(* CODESYS project Proj_3Conveyors_-_Codesys_SP19_RECOVERED_2025-03-27T17-36-29.project

Project tree, tasks and I/O mapping:
  Device : CODESYS Control Win V3 x64, 3S - Smart Software Solutions GmbH, version 3.5.19.20
    application Application
      libraries: Standard, 3.5.18.0 (System)
      task MainTask (cyclic, interval t#20ms, priority 1) calls PLC_PRG, SCADA_PRG
      function block Linear_Conveyor [SFC]: passRecipe, copy_recipe
      program PLC_PRG [CFC]
      function block WarehouseInConveyor [SFC]: copy_recipe
      function block Machine [SFC]: IncrementStep, sendTrans, checkOpPossible, copy_recipe, ChangeCurrTool, DefinePassedRecipe
      data type INSTRUCTION
      data type RECIPE_STRUCT
      program SCADA_PRG [ST]
      function block WarehouseOutConveyor [SFC]: copy_recipe
    Ethernet : Ethernet, CODESYS, version 4.2.0.0
      ModbusTCP_Slave_Device : ModbusTCP Slave Device, 3S - Smart Software Solutions GmbH, version 4.3.0.0
          settings: UpdateableHolding = TRUE; DistinctBitAreas = TRUE; Coils Size = 8; Discrete Inputs Size = 8
          output S_sensor1 : BOOL  // Holding Registers.Holding Registers.Bit0
          output S_sensor2 : BOOL  // Holding Registers.Holding Registers.Bit1
          output S_sensor3 : BOOL  // Holding Registers.Holding Registers.Bit2
          output C1_stop : BOOL  // Holding Registers.Holding Registers.Bit0
          output C2_stop : BOOL  // Holding Registers.Holding Registers.Bit1
          output C3_stop : BOOL  // Holding Registers.Holding Registers.Bit2
          output Gate0 : BOOL  // Coils.Coils.Bit0
          output Gate1 : BOOL  // Coils.Coils.Bit1
          output Gate2 : BOOL  // Coils.Coils.Bit2
          unmapped channels: Holding Registers, Input Registers, Coils, Discrete Inputs
      Modbus_TCP_Master : Modbus TCP Master, 3S - Smart Software Solutions GmbH, version 4.3.0.0
          settings: AutoReconnect = TRUE
        Modbus_TCP_Slave : Modbus TCP Slave, 3S - Smart Software Solutions GmbH, version 4.1.0.0
            settings: Unit-ID = 255; IPAddress = [127, 0, 0, 1]; Port = 5502; Channel 0.Function Code = 2; Channel 0.Read Offset = 16#0000; Channel 0.Read Length = 100; Channel 0.Write Offset = 0; Channel 0.Write Length = 0; Channel 0.Cycle Time = 100; Channel 1.Function Code = 15; Channel 1.Read Offset = 0; Channel 1.Read Length = 0; Channel 1.Write Offset = 16#0000; Channel 1.Write Length = 100; Channel 1.Cycle Time = 100
            input  Cin1_Sensor : BOOL  // Channel 0.Channel 0.Bit0
            input  Cin2_Sensor : BOOL  // Channel 0.Channel 0.Bit1
            input  Cin3_Sensor : BOOL  // Channel 0.Channel 0.Bit2
            input  Cin4_Sensor : BOOL  // Channel 0.Channel 0.Bit3
            input  AT1_in0_Sensor : BOOL  // Channel 0.Channel 0.Bit4
            input  AT1_in1_Sensor : BOOL  // Channel 0.Channel 0.Bit5
            input  AT1_in2_Sensor : BOOL  // Channel 0.Channel 0.Bit6
            input  AT1_in3_Sensor : BOOL  // Channel 0.Channel 0.Bit7
            input  AT1_in4_Sensor : BOOL  // Channel 0.Channel 0.Bit0
            input  AT1_out1_Sensor : BOOL  // Channel 0.Channel 0.Bit1
            input  AT1_out2_Sensor : BOOL  // Channel 0.Channel 0.Bit2
            input  AT1_out3_Sensor : BOOL  // Channel 0.Channel 0.Bit3
            input  AT1_out4_Sensor : BOOL  // Channel 0.Channel 0.Bit4
            input  AT1_out5_Sensor : BOOL  // Channel 0.Channel 0.Bit5
            input  AT1_out6_Sensor : BOOL  // Channel 0.Channel 0.Bit6
            input  AT2_out0_Sensor : BOOL  // Channel 0.Channel 0.Bit7
            input  AT2_out1_Sensor : BOOL  // Channel 0.Channel 0.Bit0
            input  AT2_out2_Sensor : BOOL  // Channel 0.Channel 0.Bit1
            input  AT2_out3_Sensor : BOOL  // Channel 0.Channel 0.Bit2
            input  AT2_out4_Sensor : BOOL  // Channel 0.Channel 0.Bit3
            input  AT2_in1_Sensor : BOOL  // Channel 0.Channel 0.Bit4
            input  AT2_in2_Sensor : BOOL  // Channel 0.Channel 0.Bit5
            input  AT2_in3_Sensor : BOOL  // Channel 0.Channel 0.Bit6
            input  AT2_in4_Sensor : BOOL  // Channel 0.Channel 0.Bit7
            input  AT2_in5_Sensor : BOOL  // Channel 0.Channel 0.Bit0
            input  AT2_in6_Sensor : BOOL  // Channel 0.Channel 0.Bit1
            input  Cell0_Ctop_Sensor : BOOL  // Channel 0.Channel 0.Bit2
            input  Cell0_Cmid_Sensor : BOOL  // Channel 0.Channel 0.Bit3
            input  Cell0_Cbot_Sensor : BOOL  // Channel 0.Channel 0.Bit4
            input  Cell1_Mtop_Sensor : BOOL  // Channel 0.Channel 0.Bit5
            input  Cell1_Mtop_Tool_Sensor : BOOL  // Channel 0.Channel 0.Bit6
            input  Cell1_Mtop_Y_minus_Sensor : BOOL  // Channel 0.Channel 0.Bit7
            input  Cell1_Mtop_Y_plus_Sensor : BOOL  // Channel 0.Channel 0.Bit0
            input  Cell1_Mtop_Z_minus_Sensor : BOOL  // Channel 0.Channel 0.Bit1
            input  Cell1_Mtop_Z_plus_Sensor : BOOL  // Channel 0.Channel 0.Bit2
            input  Cell1_Cmid_Sensor : BOOL  // Channel 0.Channel 0.Bit3
            input  Cell1_Mbot_Sensor : BOOL  // Channel 0.Channel 0.Bit4
            input  Cell1_Mbot_Tool_Sensor : BOOL  // Channel 0.Channel 0.Bit5
            input  Cell1_Mbot_Y_minus_Sensor : BOOL  // Channel 0.Channel 0.Bit6
            input  Cell1_Mbot_Y_plus_Sensor : BOOL  // Channel 0.Channel 0.Bit7
            input  Cell1_Mbot_Z_minus_Sensor : BOOL  // Channel 0.Channel 0.Bit0
            input  Cell1_Mbot_Z_plus_Sensor : BOOL  // Channel 0.Channel 0.Bit1
            input  Cell2_Mtop_Sensor : BOOL  // Channel 0.Channel 0.Bit2
            input  Cell2_Mtop_Tool_Sensor : BOOL  // Channel 0.Channel 0.Bit3
            input  Cell2_Mtop_Y_minus_Sensor : BOOL  // Channel 0.Channel 0.Bit4
            input  Cell2_Mtop_Y_plus_Sensor : BOOL  // Channel 0.Channel 0.Bit5
            input  Cell2_Mtop_Z_minus_Sensor : BOOL  // Channel 0.Channel 0.Bit6
            input  Cell2_Mtop_Z_plus_Sensor : BOOL  // Channel 0.Channel 0.Bit7
            input  Cell2_Cmid_Sensor : BOOL  // Channel 0.Channel 0.Bit0
            input  Cell2_Mbot_Sensor : BOOL  // Channel 0.Channel 0.Bit1
            input  Cell2_Mbot_Tool_Sensor : BOOL  // Channel 0.Channel 0.Bit2
            input  Cell2_Mbot_Y_minus_Sensor : BOOL  // Channel 0.Channel 0.Bit3
            input  Cell2_Mbot_Y_plus_Sensor : BOOL  // Channel 0.Channel 0.Bit4
            input  Cell2_Mbot_Z_minus_Sensor : BOOL  // Channel 0.Channel 0.Bit5
            input  Cell2_Mbot_Z_plus_Sensor : BOOL  // Channel 0.Channel 0.Bit6
            input  Cell3_Mtop_Sensor : BOOL  // Channel 0.Channel 0.Bit7
            input  Cell3_Mtop_Tool_Sensor : BOOL  // Channel 0.Channel 0.Bit0
            input  Cell3_Mtop_Y_minus_Sensor : BOOL  // Channel 0.Channel 0.Bit1
            input  Cell3_Mtop_Y_plus_Sensor : BOOL  // Channel 0.Channel 0.Bit2
            input  Cell3_Mtop_Z_minus_Sensor : BOOL  // Channel 0.Channel 0.Bit3
            input  Cell3_Mtop_Z_plus_Sensor : BOOL  // Channel 0.Channel 0.Bit4
            input  Cell3_Cmid_Sensor : BOOL  // Channel 0.Channel 0.Bit5
            input  Cell3_Mbot_Sensor : BOOL  // Channel 0.Channel 0.Bit6
            input  Cell3_Mbot_Tool_Sensor : BOOL  // Channel 0.Channel 0.Bit7
            input  Cell3_Mbot_Y_minus_Sensor : BOOL  // Channel 0.Channel 0.Bit0
            input  Cell3_Mbot_Y_plus_Sensor : BOOL  // Channel 0.Channel 0.Bit1
            input  Cell3_Mbot_Z_minus_Sensor : BOOL  // Channel 0.Channel 0.Bit2
            input  Cell3_Mbot_Z_plus_Sensor : BOOL  // Channel 0.Channel 0.Bit3
            input  Cell4_Mtop_Sensor : BOOL  // Channel 0.Channel 0.Bit4
            input  Cell4_Mtop_Tool_Sensor : BOOL  // Channel 0.Channel 0.Bit5
            input  Cell4_Mtop_Y_minus_Sensor : BOOL  // Channel 0.Channel 0.Bit6
            input  Cell4_Mtop_Y_plus_Sensor : BOOL  // Channel 0.Channel 0.Bit7
            input  Cell4_Mtop_Z_minus_Sensor : BOOL  // Channel 0.Channel 0.Bit0
            input  Cell4_Mtop_Z_plus_Sensor : BOOL  // Channel 0.Channel 0.Bit1
            input  Cell4_Cmid_Sensor : BOOL  // Channel 0.Channel 0.Bit2
            input  Cell4_Mbot_Sensor : BOOL  // Channel 0.Channel 0.Bit3
            input  Cell4_Mbot_Tool_Sensor : BOOL  // Channel 0.Channel 0.Bit4
            input  Cell4_Mbot_Y_minus_Sensor : BOOL  // Channel 0.Channel 0.Bit5
            input  Cell4_Mbot_Y_plus_Sensor : BOOL  // Channel 0.Channel 0.Bit6
            input  Cell4_Mbot_Z_minus_Sensor : BOOL  // Channel 0.Channel 0.Bit7
            input  Cell4_Mbot_Z_plus_Sensor : BOOL  // Channel 0.Channel 0.Bit0
            input  Cell5_Mtop_Sensor : BOOL  // Channel 0.Channel 0.Bit1
            input  Cell5_Mtop_Tool_Sensor : BOOL  // Channel 0.Channel 0.Bit2
            input  Cell5_Mtop_Y_minus_Sensor : BOOL  // Channel 0.Channel 0.Bit3
            input  Cell5_Mtop_Y_plus_Sensor : BOOL  // Channel 0.Channel 0.Bit4
            input  Cell5_Mtop_Z_minus_Sensor : BOOL  // Channel 0.Channel 0.Bit5
            input  Cell5_Mtop_Z_plus_Sensor : BOOL  // Channel 0.Channel 0.Bit6
            input  Cell5_Cmid_Sensor : BOOL  // Channel 0.Channel 0.Bit7
            input  Cell5_Mbot_Sensor : BOOL  // Channel 0.Channel 0.Bit0
            input  Cell5_Mbot_Tool_Sensor : BOOL  // Channel 0.Channel 0.Bit1
            input  Cell5_Mbot_Y_minus_Sensor : BOOL  // Channel 0.Channel 0.Bit2
            input  Cell5_Mbot_Y_plus_Sensor : BOOL  // Channel 0.Channel 0.Bit3
            input  Cell5_Mbot_Z_minus_Sensor : BOOL  // Channel 0.Channel 0.Bit4
            input  Cell5_Mbot_Z_plus_Sensor : BOOL  // Channel 0.Channel 0.Bit5
            input  Cell6_Mtop_Sensor : BOOL  // Channel 0.Channel 0.Bit6
            input  Cell6_Mtop_Tool_Sensor : BOOL  // Channel 0.Channel 0.Bit7
            input  Cell6_Mtop_Y_minus_Sensor : BOOL  // Channel 0.Channel 0.Bit0
            input  Cell6_Mtop_Y_plus_Sensor : BOOL  // Channel 0.Channel 0.Bit1
            input  Cell6_Mtop_Z_minus_Sensor : BOOL  // Channel 0.Channel 0.Bit2
            input  Cell6_Mtop_Z_plus_Sensor : BOOL  // Channel 0.Channel 0.Bit3
            output Cin1_Motor_plus : BOOL  // Channel 1.Channel 1.Bit0
            output Cin1_Motor_minus : BOOL  // Channel 1.Channel 1.Bit1
            output Cin2_Motor_plus : BOOL  // Channel 1.Channel 1.Bit2
            output Cin2_Motor_minus : BOOL  // Channel 1.Channel 1.Bit3
            output Cin3_Motor_plus : BOOL  // Channel 1.Channel 1.Bit4
            output Cin3_Motor_minus : BOOL  // Channel 1.Channel 1.Bit5
            output Cin4_Motor_plus : BOOL  // Channel 1.Channel 1.Bit6
            output Cin4_Motor_minus : BOOL  // Channel 1.Channel 1.Bit7
            output AT1_in0_Motor_plus : BOOL  // Channel 1.Channel 1.Bit0
            output AT1_in0_Motor_minus : BOOL  // Channel 1.Channel 1.Bit1
            output AT1_in0_Warehouse_In : BOOL  // Channel 1.Channel 1.Bit2
            output AT1_in1_Motor_plus : BOOL  // Channel 1.Channel 1.Bit3
            output AT1_in1_Motor_minus : BOOL  // Channel 1.Channel 1.Bit4
            output AT1_in1_Warehouse_In : BOOL  // Channel 1.Channel 1.Bit5
            output AT1_in2_Motor_plus : BOOL  // Channel 1.Channel 1.Bit6
            output AT1_in2_Motor_minus : BOOL  // Channel 1.Channel 1.Bit7
            output AT1_in2_Warehouse_In : BOOL  // Channel 1.Channel 1.Bit0
            output AT1_in3_Motor_plus : BOOL  // Channel 1.Channel 1.Bit1
            output AT1_in3_Motor_minus : BOOL  // Channel 1.Channel 1.Bit2
            output AT1_in3_Warehouse_In : BOOL  // Channel 1.Channel 1.Bit3
            output AT1_in4_Motor_plus : BOOL  // Channel 1.Channel 1.Bit4
            output AT1_in4_Motor_minus : BOOL  // Channel 1.Channel 1.Bit5
            output AT1_in4_Warehouse_In : BOOL  // Channel 1.Channel 1.Bit6
            output AT1_out1_Motor_plus : BOOL  // Channel 1.Channel 1.Bit7
            output AT1_out1_Motor_minus : BOOL  // Channel 1.Channel 1.Bit0
            output AT1_out2_Motor_plus : BOOL  // Channel 1.Channel 1.Bit1
            output AT1_out2_Motor_minus : BOOL  // Channel 1.Channel 1.Bit2
            output AT1_out3_Motor_plus : BOOL  // Channel 1.Channel 1.Bit3
            output AT1_out3_Motor_minus : BOOL  // Channel 1.Channel 1.Bit4
            output AT1_out4_Motor_plus : BOOL  // Channel 1.Channel 1.Bit5
            output AT1_out4_Motor_minus : BOOL  // Channel 1.Channel 1.Bit6
            output AT1_out5_Motor_plus : BOOL  // Channel 1.Channel 1.Bit7
            output AT1_out5_Motor_minus : BOOL  // Channel 1.Channel 1.Bit0
            output AT1_out6_Motor_plus : BOOL  // Channel 1.Channel 1.Bit1
            output AT1_out6_Motor_minus : BOOL  // Channel 1.Channel 1.Bit2
            output AT2_out0_Motor_plus : BOOL  // Channel 1.Channel 1.Bit3
            output AT2_out0_Motor_minus : BOOL  // Channel 1.Channel 1.Bit4
            output AT2_out1_Motor_plus : BOOL  // Channel 1.Channel 1.Bit5
            output AT2_out1_Motor_minus : BOOL  // Channel 1.Channel 1.Bit6
            output AT2_out2_Motor_plus : BOOL  // Channel 1.Channel 1.Bit7
            output AT2_out2_Motor_minus : BOOL  // Channel 1.Channel 1.Bit0
            output AT2_out3_Motor_plus : BOOL  // Channel 1.Channel 1.Bit1
            output AT2_out3_Motor_minus : BOOL  // Channel 1.Channel 1.Bit2
            output AT2_out4_Motor_plus : BOOL  // Channel 1.Channel 1.Bit3
            output AT2_out4_Motor_minus : BOOL  // Channel 1.Channel 1.Bit4
            output AT2_in1_Motor_plus : BOOL  // Channel 1.Channel 1.Bit5
            output AT2_in1_Motor_minus : BOOL  // Channel 1.Channel 1.Bit6
            output AT2_in1_Warehouse_In : BOOL  // Channel 1.Channel 1.Bit7
            output AT2_in2_Motor_plus : BOOL  // Channel 1.Channel 1.Bit0
            output AT2_in2_Motor_minus : BOOL  // Channel 1.Channel 1.Bit1
            output AT2_in2_Warehouse_In : BOOL  // Channel 1.Channel 1.Bit2
            output AT2_in3_Motor_plus : BOOL  // Channel 1.Channel 1.Bit3
            output AT2_in3_Motor_minus : BOOL  // Channel 1.Channel 1.Bit4
            output AT2_in3_Warehouse_In : BOOL  // Channel 1.Channel 1.Bit5
            output AT2_in4_Motor_plus : BOOL  // Channel 1.Channel 1.Bit6
            output AT2_in4_Motor_minus : BOOL  // Channel 1.Channel 1.Bit7
            output AT2_in4_Warehouse_In : BOOL  // Channel 1.Channel 1.Bit0
            output AT2_in5_Motor_plus : BOOL  // Channel 1.Channel 1.Bit1
            output AT2_in5_Motor_minus : BOOL  // Channel 1.Channel 1.Bit2
            output AT2_in5_Warehouse_In : BOOL  // Channel 1.Channel 1.Bit3
            output AT2_in6_Motor_plus : BOOL  // Channel 1.Channel 1.Bit4
            output AT2_in6_Motor_minus : BOOL  // Channel 1.Channel 1.Bit5
            output AT2_in6_Warehouse_In : BOOL  // Channel 1.Channel 1.Bit6
            output Cell0_Ctop_Motor_plus : BOOL  // Channel 1.Channel 1.Bit7
            output Cell0_Ctop_Motor_minus : BOOL  // Channel 1.Channel 1.Bit0
            output Cell0_Cmid_Motor_plus : BOOL  // Channel 1.Channel 1.Bit1
            output Cell0_Cmid_Motor_minus : BOOL  // Channel 1.Channel 1.Bit2
            output Cell0_Cbot_Motor_plus : BOOL  // Channel 1.Channel 1.Bit3
            output Cell0_Cbot_Motor_minus : BOOL  // Channel 1.Channel 1.Bit4
            output Cell1_Mtop_Motor_plus : BOOL  // Channel 1.Channel 1.Bit5
            output Cell1_Mtop_Motor_minus : BOOL  // Channel 1.Channel 1.Bit6
            output Cell1_Mtop_Rotate_minus : BOOL  // Channel 1.Channel 1.Bit7
            output Cell1_Mtop_Rotate_plus : BOOL  // Channel 1.Channel 1.Bit0
            output Cell1_Mtop_Tool : BOOL  // Channel 1.Channel 1.Bit1
            output Cell1_Mtop_Y_minus : BOOL  // Channel 1.Channel 1.Bit2
            output Cell1_Mtop_Y_plus : BOOL  // Channel 1.Channel 1.Bit3
            output Cell1_Mtop_Z_minus : BOOL  // Channel 1.Channel 1.Bit4
            output Cell1_Mtop_Z_plus : BOOL  // Channel 1.Channel 1.Bit5
            output Cell1_Cmid_Motor_plus : BOOL  // Channel 1.Channel 1.Bit6
            output Cell1_Cmid_Motor_minus : BOOL  // Channel 1.Channel 1.Bit7
            output Cell1_Mbot_Motor_plus : BOOL  // Channel 1.Channel 1.Bit0
            output Cell1_Mbot_Motor_minus : BOOL  // Channel 1.Channel 1.Bit1
            output Cell1_Mbot_Rotate_minus : BOOL  // Channel 1.Channel 1.Bit2
            output Cell1_Mbot_Rotate_plus : BOOL  // Channel 1.Channel 1.Bit3
            output Cell1_Mbot_Tool : BOOL  // Channel 1.Channel 1.Bit4
            output Cell1_Mbot_Y_minus : BOOL  // Channel 1.Channel 1.Bit5
            output Cell1_Mbot_Y_plus : BOOL  // Channel 1.Channel 1.Bit6
            output Cell1_Mbot_Z_minus : BOOL  // Channel 1.Channel 1.Bit7
            output Cell1_Mbot_Z_plus : BOOL  // Channel 1.Channel 1.Bit0
            output Cell2_Mtop_Motor_plus : BOOL  // Channel 1.Channel 1.Bit1
            output Cell2_Mtop_Motor_minus : BOOL  // Channel 1.Channel 1.Bit2
            output Cell2_Mtop_Rotate_minus : BOOL  // Channel 1.Channel 1.Bit3
            output Cell2_Mtop_Rotate_plus : BOOL  // Channel 1.Channel 1.Bit4
            output Cell2_Mtop_Tool : BOOL  // Channel 1.Channel 1.Bit5
            output Cell2_Mtop_Y_minus : BOOL  // Channel 1.Channel 1.Bit6
            output Cell2_Mtop_Y_plus : BOOL  // Channel 1.Channel 1.Bit7
            output Cell2_Mtop_Z_minus : BOOL  // Channel 1.Channel 1.Bit0
            output Cell2_Mtop_Z_plus : BOOL  // Channel 1.Channel 1.Bit1
            output Cell2_Cmid_Motor_plus : BOOL  // Channel 1.Channel 1.Bit2
            output Cell2_Cmid_Motor_minus : BOOL  // Channel 1.Channel 1.Bit3
            unmapped channels: Channel 0, Channel 1
*)

// Device/Application/INSTRUCTION
TYPE INSTRUCTION :
STRUCT
	tool: INT;
	process_time: TIME;
END_STRUCT
END_TYPE

// Device/Application/RECIPE_STRUCT
TYPE RECIPE_STRUCT :
STRUCT
	Piece: INT;
	Instruction_list: ARRAY[1..3] OF INSTRUCTION;
	Step: INT;
END_STRUCT
END_TYPE

// Device/Application/PLC_PRG
PROGRAM PLC_PRG
VAR
	C1, C2, C3: Linear_Conveyor;
	M1,M2: Machine;
	WC1: WarehouseInConveyor;
	
	M1_tools : ARRAY[1..3] OF INT := [1,2,3];
	M2_tools : ARRAY[1..3] OF INT := [4,5,6];
	
	test_instruction : INSTRUCTION := (tool := 1, process_time :=T#20S);
	test_instruction2 : INSTRUCTION := (tool := 5, process_time :=T#30S);
	test_array : ARRAY [1..3] OF INSTRUCTION := [test_instruction,test_instruction2,test_instruction];
	
	test_recipe : RECIPE_STRUCT := (Piece:=1, Instruction_list := test_array ,Step:=1);
	
	WCO1: WarehouseOutConveyor;
END_VAR

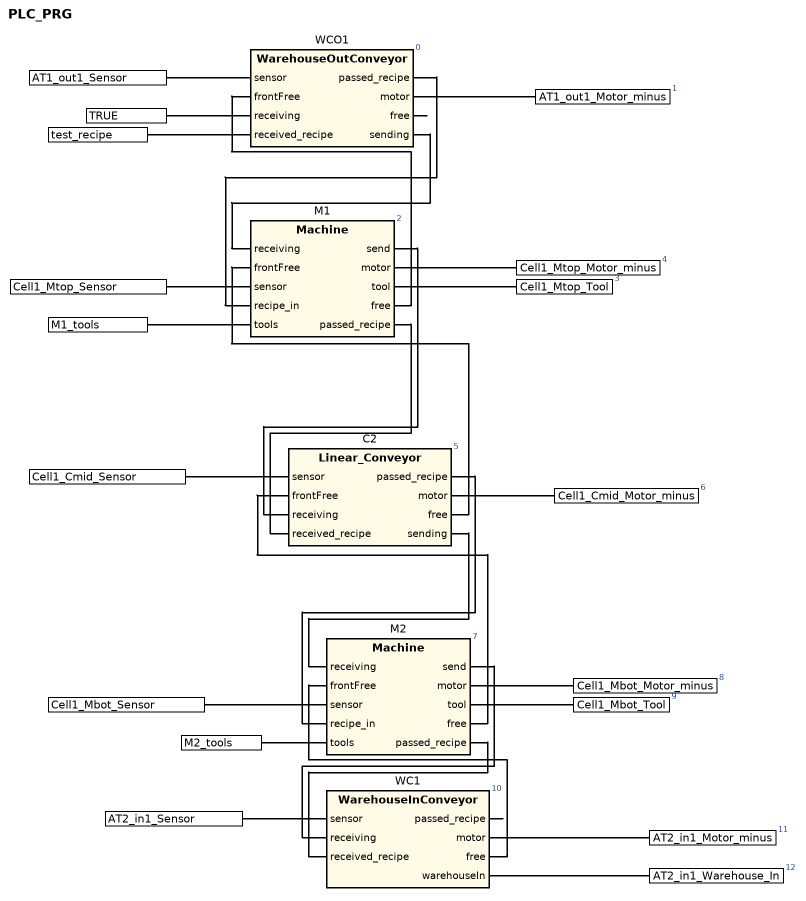
WCO1(sensor := AT1_out1_Sensor, frontFree := M1.free, receiving := TRUE, received_recipe := test_recipe); // WarehouseOutConveyor
AT1_out1_Motor_minus := WCO1.motor;
M1(
    receiving := WCO1.sending,
    frontFree := C2.free,
    sensor := Cell1_Mtop_Sensor,
    recipe_in := WCO1.passed_recipe,
    tools := M1_tools); // Machine
Cell1_Mtop_Tool := M1.tool;
Cell1_Mtop_Motor_minus := M1.motor;
C2(
    sensor := Cell1_Cmid_Sensor,
    frontFree := M2.free,
    receiving := M1.send,
    received_recipe := M1.passed_recipe); // Linear_Conveyor
Cell1_Cmid_Motor_minus := C2.motor;
M2(
    receiving := C2.sending,
    frontFree := WC1.free,
    sensor := Cell1_Mbot_Sensor,
    recipe_in := C2.passed_recipe,
    tools := M2_tools); // Machine
Cell1_Mbot_Motor_minus := M2.motor;
Cell1_Mbot_Tool := M2.tool;
WC1(sensor := AT2_in1_Sensor, receiving := M2.send, received_recipe := M2.passed_recipe); // WarehouseInConveyor
AT2_in1_Motor_minus := WC1.motor;
AT2_in1_Warehouse_In := WC1.warehouseIn;

END_PROGRAM

// Device/Application/WarehouseInConveyor
FUNCTION_BLOCK WarehouseInConveyor
VAR_INPUT
	sensor: BOOL;
	receiving: BOOL;
	received_recipe : RECIPE_STRUCT;
END_VAR
VAR_OUTPUT
	passed_recipe : RECIPE_STRUCT := received_recipe;
	motor : BOOL;
	free: BOOL;
	warehouseIn: BOOL;
END_VAR
VAR
END_VAR

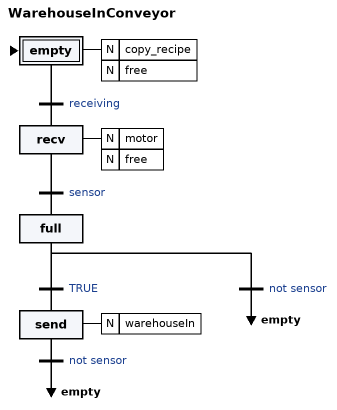
INITIAL_STEP empty:
    copy_recipe(N);
    free(N);
END_STEP
TRANSITION FROM empty TO recv
    := receiving;
END_TRANSITION
STEP recv:
    motor(N);
    free(N);
END_STEP
TRANSITION FROM recv TO full
    := sensor;
END_TRANSITION
STEP full:
END_STEP
TRANSITION FROM full TO send
    := TRUE;
END_TRANSITION
TRANSITION FROM full TO empty
    := not sensor;
END_TRANSITION
STEP send:
    warehouseIn(N);
END_STEP
TRANSITION FROM send TO empty
    := not sensor;
END_TRANSITION

ACTION copy_recipe:
passed_recipe:=received_recipe;
END_ACTION

END_FUNCTION_BLOCK

// Device/Application/Linear_Conveyor
FUNCTION_BLOCK Linear_Conveyor
VAR_INPUT
	sensor: BOOL;
	frontFree: BOOL;
	receiving: BOOL;
	received_recipe : RECIPE_STRUCT;
END_VAR
VAR_OUTPUT
	passed_recipe : RECIPE_STRUCT := received_recipe;
	motor : BOOL;
	free: BOOL;
	sending: BOOL;
END_VAR
VAR
END_VAR

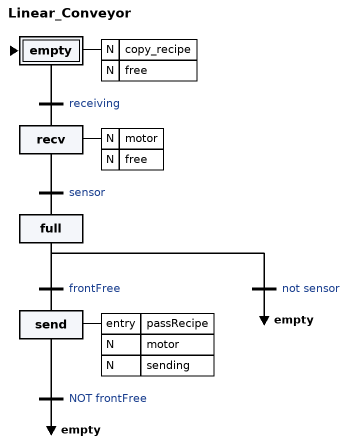
INITIAL_STEP empty:
    copy_recipe(N);
    free(N);
END_STEP
TRANSITION FROM empty TO recv
    := receiving;
END_TRANSITION
STEP recv:
    motor(N);
    free(N);
END_STEP
TRANSITION FROM recv TO full
    := sensor;
END_TRANSITION
STEP full:
END_STEP
TRANSITION FROM full TO send
    := frontFree;
END_TRANSITION
TRANSITION FROM full TO empty
    := not sensor;
END_TRANSITION
STEP send:
    passRecipe(P1);  // entry action
    motor(N);
    sending(N);
END_STEP
TRANSITION FROM send TO empty
    := NOT frontFree;
END_TRANSITION

ACTION passRecipe:
passed_recipe:=received_recipe;
END_ACTION

ACTION copy_recipe:
passed_recipe := received_recipe;
END_ACTION

END_FUNCTION_BLOCK

// Device/Application/WarehouseOutConveyor
FUNCTION_BLOCK WarehouseOutConveyor
VAR_INPUT
	sensor: BOOL;
	frontFree: BOOL;
	receiving: BOOL;
	received_recipe : RECIPE_STRUCT;
END_VAR
VAR_OUTPUT
	passed_recipe : RECIPE_STRUCT := received_recipe;
	motor : BOOL;
	free: BOOL;
	sending: BOOL;
END_VAR
VAR
END_VAR

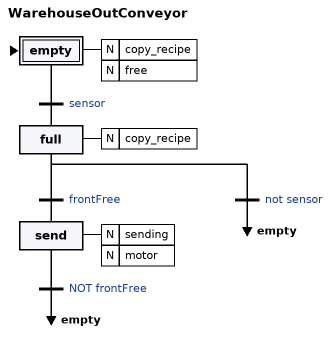
INITIAL_STEP empty:
    copy_recipe(N);
    free(N);
END_STEP
TRANSITION FROM empty TO full
    := sensor;
END_TRANSITION
STEP full:
    copy_recipe(N);
END_STEP
TRANSITION FROM full TO send
    := frontFree;
END_TRANSITION
TRANSITION FROM full TO empty
    := not sensor;
END_TRANSITION
STEP send:
    sending(N);
    motor(N);
END_STEP
TRANSITION FROM send TO empty
    := NOT frontFree;
END_TRANSITION

ACTION copy_recipe:
passed_recipe:=received_recipe;
END_ACTION

END_FUNCTION_BLOCK

// Device/Application/Machine
FUNCTION_BLOCK Machine
VAR_INPUT
	receiving:BOOL;
	frontFree:BOOL;
	sensor:BOOL;
	recipe_in: RECIPE_STRUCT;
	tools: ARRAY[1..3] OF INT;
END_VAR
VAR_OUTPUT
	send:BOOL;
	motor:BOOL;
	tool:BOOL;
	free:BOOL;
	passed_recipe : RECIPE_STRUCT;
END_VAR
VAR
	timeForChange : TIME := T#30s;
	opPossible:BOOL:=FALSE;
	currTool:INT:=1;
	i:INT;
	steps_done : INT := 0;
	currToolIsTool : BOOL := FALSE;
	recipe : RECIPE_STRUCT;
	manualMode: BOOL;
END_VAR

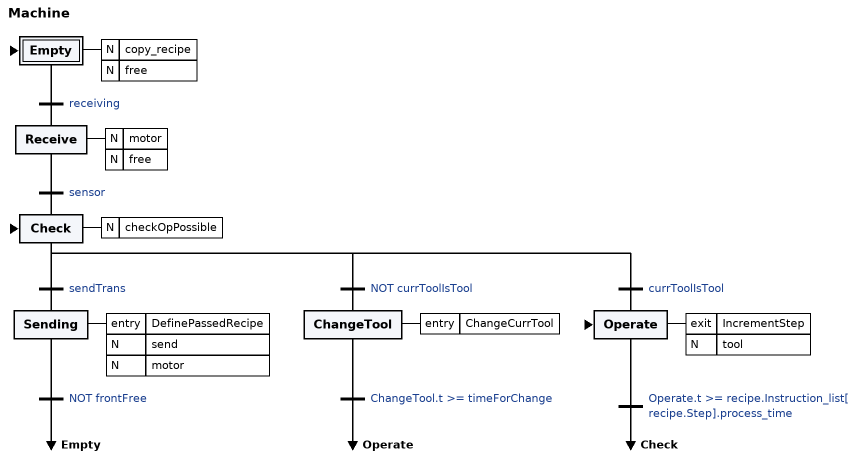
INITIAL_STEP Empty:
    copy_recipe(N);
    free(N);
END_STEP
TRANSITION FROM Empty TO Receive
    := receiving;
END_TRANSITION
STEP Receive:
    motor(N);
    free(N);
END_STEP
TRANSITION FROM Receive TO Check
    := sensor;
END_TRANSITION
STEP Check:
    checkOpPossible(N);
END_STEP
TRANSITION FROM Check TO Sending
    := sendTrans;
END_TRANSITION
STEP Sending:
    DefinePassedRecipe(P1);  // entry action
    send(N);
    motor(N);
END_STEP
TRANSITION FROM Sending TO Empty
    := NOT frontFree;
END_TRANSITION
TRANSITION FROM Check TO ChangeTool
    := NOT currToolIsTool;
END_TRANSITION
STEP ChangeTool:
    ChangeCurrTool(P1);  // entry action
END_STEP
TRANSITION FROM ChangeTool TO Operate
    := ChangeTool.t >= timeForChange;
END_TRANSITION
TRANSITION FROM Check TO Operate
    := currToolIsTool;
END_TRANSITION
STEP Operate:
    IncrementStep(P0);  // exit action
    tool(N);
END_STEP
TRANSITION FROM Operate TO Check
    := Operate.t >= recipe.Instruction_list[recipe.Step].process_time;
END_TRANSITION

ACTION IncrementStep:
steps_done := steps_done + 1;
END_ACTION

TRANSITION sendTrans:
sendTrans:= (NOT opPossible) AND (frontFree);
END_TRANSITION

ACTION checkOpPossible:
opPossible:=FALSE;
IF (recipe.Step + steps_done) <= 3 THEN
	FOR i := 1 TO 3 DO
		IF recipe.Instruction_list[recipe.Step + steps_done].tool = tools[i] THEN
			opPossible:=TRUE;
		END_IF
	END_FOR;
END_IF

currToolIsTool := opPossible AND (currTool=recipe.Instruction_list[recipe.Step].tool);
END_ACTION

ACTION copy_recipe:
recipe := recipe_in;
passed_recipe := recipe;
passed_recipe.Step := passed_recipe.Step+steps_done;
END_ACTION

ACTION ChangeCurrTool:
currTool := recipe.Instruction_list[recipe.Step].tool;
END_ACTION

ACTION DefinePassedRecipe:
passed_recipe := recipe;
passed_recipe.Step:=recipe.Step+steps_done;
END_ACTION

END_FUNCTION_BLOCK

// Device/Application/SCADA_PRG
PROGRAM SCADA_PRG
VAR
END_VAR

END_PROGRAM
